{attribute 'GeneratedUsingTerminal: KL6211-0022'}
{attribute addProperty BoxType "KL6211-0022"}
{attribute addProperty Id "Channel_1AT %Q*Channel_332F026B0"}
{attribute addProperty CRC "1234012259"}
{attribute addProperty Size "0"}
TYPE KL_498D8863 :
STRUCT
	{attribute addProperty Name "Channel_1"}
	Channel_1 : Channel_332F026B;
END_STRUCT
END_TYPE

(* stored: Version 1.2.0.0, ProductVersion 3.1.4024.9
   DUT KL_498D8863: Id {d8840a87-7c97-463f-ad6a-fe8efca4014a} *)
